REGION Network 79: Coordination Out - Decoilers Horizontal Rotation
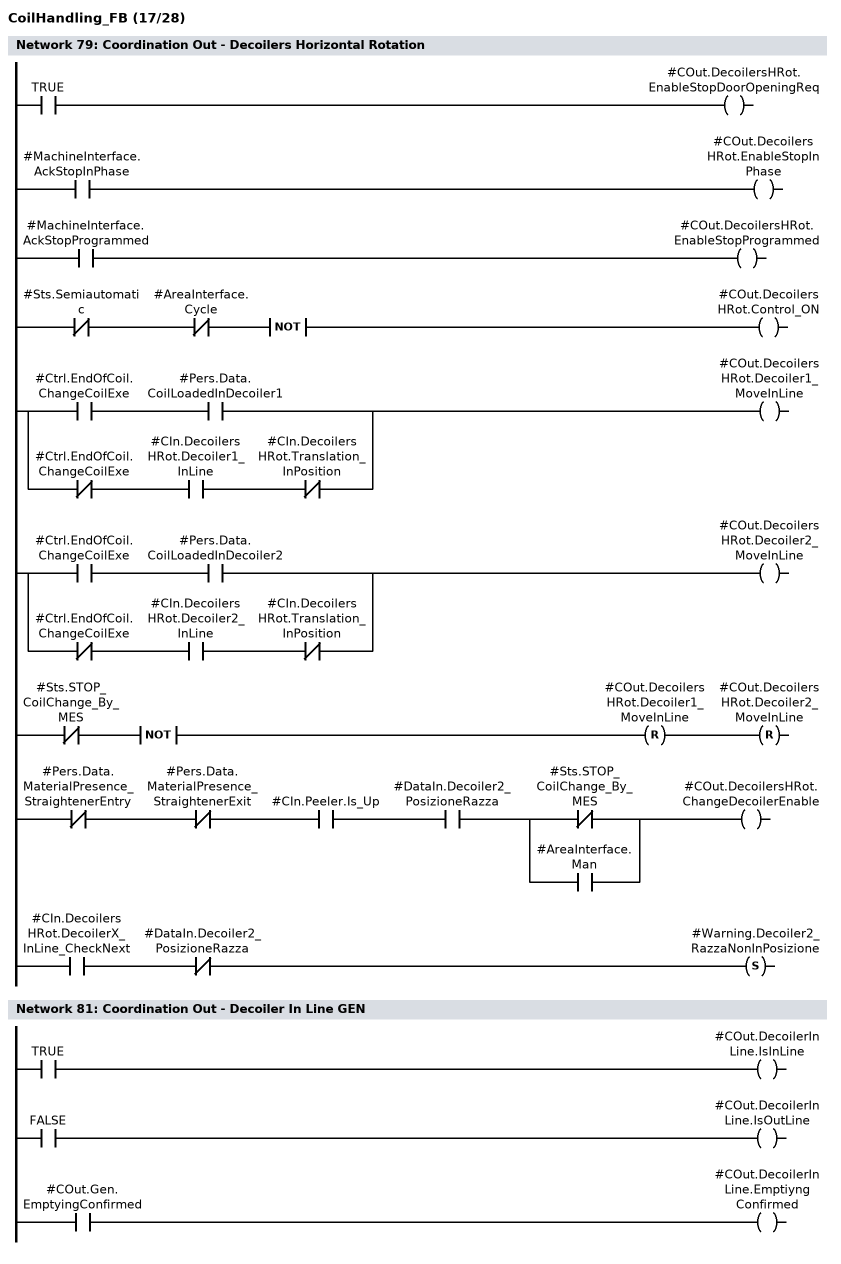
   RUNG wire#powerrail
      Contact( TRUE )
      Coil( #COut.DecoilersHRot.EnableStopDoorOpeningReq )
   END_RUNG
   RUNG wire#powerrail
      Contact( #MachineInterface.AckStopInPhase )
      Coil( #COut.DecoilersHRot.EnableStopInPhase )
   END_RUNG
   RUNG wire#powerrail
      Contact( #MachineInterface.AckStopProgrammed )
      Coil( #COut.DecoilersHRot.EnableStopProgrammed )
   END_RUNG
   RUNG wire#powerrail
      I_Contact( #Sts.Semiautomatic )
      I_Contact( #AreaInterface.Cycle )
      Not()
      Coil( #COut.DecoilersHRot.Control_ON )
   END_RUNG
   RUNG wire#powerrail
      Contact( #Ctrl.EndOfCoil.ChangeCoilExe )
      Contact( #Pers.Data.CoilLoadedInDecoiler1 )
      wire#w1
      Coil( #COut.DecoilersHRot.Decoiler1_MoveInLine )
   END_RUNG
   RUNG wire#powerrail
      I_Contact( #Ctrl.EndOfCoil.ChangeCoilExe )
      Contact( #CIn.DecoilersHRot.Decoiler1_InLine )
      I_Contact( #CIn.DecoilersHRot.Translation_InPosition )
   END_RUNG wire#w1
   RUNG wire#powerrail
      Contact( #Ctrl.EndOfCoil.ChangeCoilExe )
      Contact( #Pers.Data.CoilLoadedInDecoiler2 )
      wire#w2
      Coil( #COut.DecoilersHRot.Decoiler2_MoveInLine )
   END_RUNG
   RUNG wire#powerrail
      I_Contact( #Ctrl.EndOfCoil.ChangeCoilExe )
      Contact( #CIn.DecoilersHRot.Decoiler2_InLine )
      I_Contact( #CIn.DecoilersHRot.Translation_InPosition )
   END_RUNG wire#w2
   RUNG wire#powerrail
      I_Contact( #Sts.STOP_CoilChange_By_MES )
      Not()
      R_Coil( #COut.DecoilersHRot.Decoiler1_MoveInLine )
      R_Coil( #COut.DecoilersHRot.Decoiler2_MoveInLine )
   END_RUNG
   RUNG wire#powerrail
      I_Contact( #Pers.Data.MaterialPresence_StraightenerEntry )
      I_Contact( #Pers.Data.MaterialPresence_StraightenerExit )
      Contact( #CIn.Peeler.Is_Up )
      Contact( #DataIn.Decoiler2_PosizioneRazza )
      wire#w3
      I_Contact( #Sts.STOP_CoilChange_By_MES )
      wire#w4
      Coil( #COut.DecoilersHRot.ChangeDecoilerEnable )
   END_RUNG
   RUNG wire#w3
      Contact( #AreaInterface.Man )
   END_RUNG wire#w4
   RUNG wire#powerrail
      Contact( #CIn.DecoilersHRot.DecoilerX_InLine_CheckNext )
      I_Contact( #DataIn.Decoiler2_PosizioneRazza )
      S_Coil( #Warning.Decoiler2_RazzaNonInPosizione )
   END_RUNG
   // the same network as SCL:
   #COut.DecoilersHRot.EnableStopDoorOpeningReq := TRUE;
   #COut.DecoilersHRot.EnableStopInPhase := #MachineInterface.AckStopInPhase;
   #COut.DecoilersHRot.EnableStopProgrammed := #MachineInterface.AckStopProgrammed;
   #COut.DecoilersHRot.Control_ON := NOT (NOT #Sts.Semiautomatic AND NOT #AreaInterface.Cycle);
   #COut.DecoilersHRot.Decoiler1_MoveInLine := (#Ctrl.EndOfCoil.ChangeCoilExe AND #Pers.Data.CoilLoadedInDecoiler1) OR (NOT #Ctrl.EndOfCoil.ChangeCoilExe AND #CIn.DecoilersHRot.Decoiler1_InLine AND NOT #CIn.DecoilersHRot.Translation_InPosition);
   #COut.DecoilersHRot.Decoiler2_MoveInLine := (#Ctrl.EndOfCoil.ChangeCoilExe AND #Pers.Data.CoilLoadedInDecoiler2) OR (NOT #Ctrl.EndOfCoil.ChangeCoilExe AND #CIn.DecoilersHRot.Decoiler2_InLine AND NOT #CIn.DecoilersHRot.Translation_InPosition);
   IF NOT (NOT #Sts.STOP_CoilChange_By_MES) THEN
       #COut.DecoilersHRot.Decoiler1_MoveInLine := FALSE;
       #COut.DecoilersHRot.Decoiler2_MoveInLine := FALSE;
   END_IF;
   #COut.DecoilersHRot.ChangeDecoilerEnable := NOT #Pers.Data.MaterialPresence_StraightenerEntry AND NOT #Pers.Data.MaterialPresence_StraightenerExit AND #CIn.Peeler.Is_Up AND #DataIn.Decoiler2_PosizioneRazza AND (NOT #Sts.STOP_CoilChange_By_MES OR #AreaInterface.Man);
   IF #CIn.DecoilersHRot.DecoilerX_InLine_CheckNext AND NOT #DataIn.Decoiler2_PosizioneRazza THEN
       #Warning.Decoiler2_RazzaNonInPosizione := TRUE;
   END_IF;
END_REGION

REGION Network 80: <+>
END_REGION

REGION Network 81: Coordination Out - Decoiler In Line GEN
   RUNG wire#powerrail
      Contact( TRUE )
      Coil( #COut.DecoilerInLine.IsInLine )
   END_RUNG
   RUNG wire#powerrail
      Contact( FALSE )
      Coil( #COut.DecoilerInLine.IsOutLine )
   END_RUNG
   RUNG wire#powerrail
      Contact( #COut.Gen.EmptyingConfirmed )
      Coil( #COut.DecoilerInLine.EmptiyngConfirmed )
   END_RUNG
   // the same network as SCL:
   #COut.DecoilerInLine.IsInLine := TRUE;
   #COut.DecoilerInLine.IsOutLine := FALSE;
   #COut.DecoilerInLine.EmptiyngConfirmed := #COut.Gen.EmptyingConfirmed;
END_REGION

REGION Network 82: Coordination Out - Decoiler in Line BRAKE
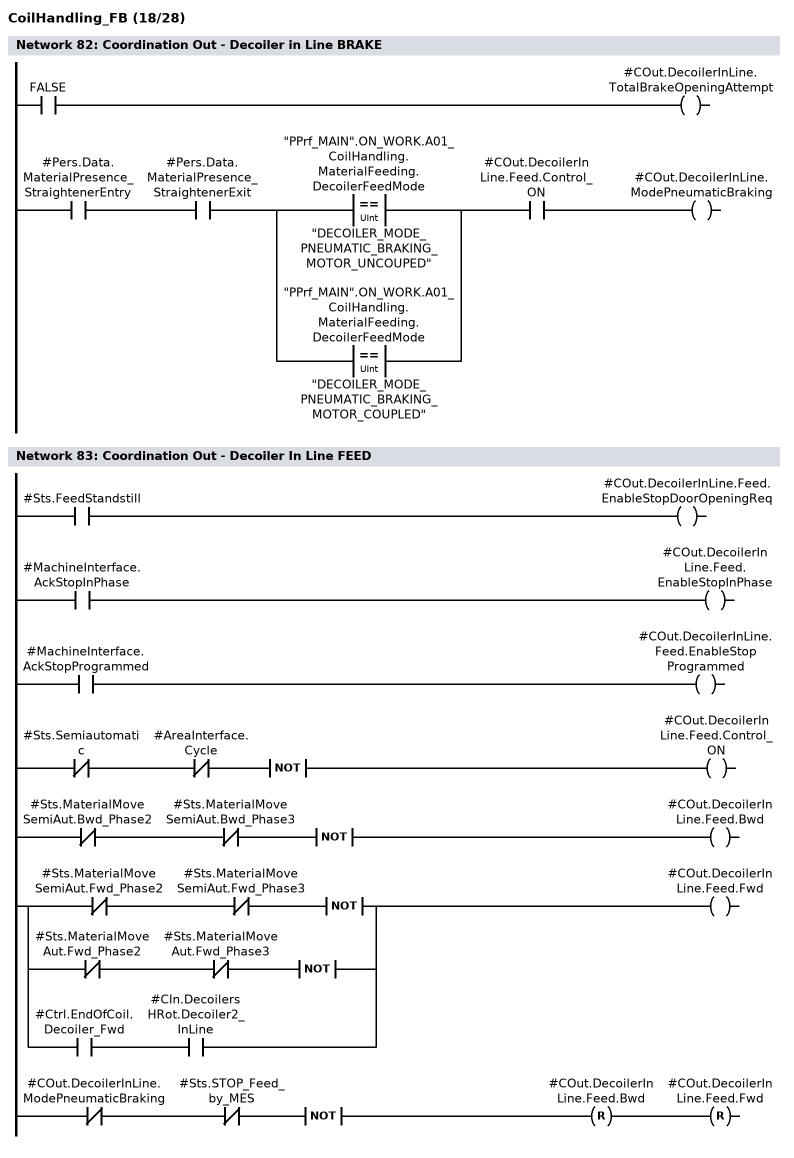
   RUNG wire#powerrail
      Contact( FALSE )
      Coil( #COut.DecoilerInLine.TotalBrakeOpeningAttempt )
   END_RUNG
   RUNG wire#powerrail
      Contact( #Pers.Data.MaterialPresence_StraightenerEntry )
      Contact( #Pers.Data.MaterialPresence_StraightenerExit )
      wire#w1
      { S7_Templates := "SrcType := UInt" } EQ_Contact(in1 := "PPrf_MAIN".ON_WORK.A01_CoilHandling.MaterialFeeding.DecoilerFeedMode, in2 := "DECOILER_MODE_PNEUMATIC_BRAKING_MOTOR_UNCOUPED")
      wire#w2
      Contact( #COut.DecoilerInLine.Feed.Control_ON )
      Coil( #COut.DecoilerInLine.ModePneumaticBraking )
   END_RUNG
   RUNG wire#w1
      { S7_Templates := "SrcType := UInt" } EQ_Contact(in1 := "PPrf_MAIN".ON_WORK.A01_CoilHandling.MaterialFeeding.DecoilerFeedMode, in2 := "DECOILER_MODE_PNEUMATIC_BRAKING_MOTOR_COUPLED")
   END_RUNG wire#w2
   // the same network as SCL:
   #COut.DecoilerInLine.TotalBrakeOpeningAttempt := FALSE;
   #COut.DecoilerInLine.ModePneumaticBraking := #Pers.Data.MaterialPresence_StraightenerEntry AND #Pers.Data.MaterialPresence_StraightenerExit AND (("PPrf_MAIN".ON_WORK.A01_CoilHandling.MaterialFeeding.DecoilerFeedMode = "DECOILER_MODE_PNEUMATIC_BRAKING_MOTOR_UNCOUPED") OR ("PPrf_MAIN".ON_WORK.A01_CoilHandling.MaterialFeeding.DecoilerFeedMode = "DECOILER_MODE_PNEUMATIC_BRAKING_MOTOR_COUPLED")) AND #COut.DecoilerInLine.Feed.Control_ON;
END_REGION

REGION Network 83: Coordination Out - Decoiler In Line FEED
   RUNG wire#powerrail
      Contact( #Sts.FeedStandstill )
      Coil( #COut.DecoilerInLine.Feed.EnableStopDoorOpeningReq )
   END_RUNG
   RUNG wire#powerrail
      Contact( #MachineInterface.AckStopInPhase )
      Coil( #COut.DecoilerInLine.Feed.EnableStopInPhase )
   END_RUNG
   RUNG wire#powerrail
      Contact( #MachineInterface.AckStopProgrammed )
      Coil( #COut.DecoilerInLine.Feed.EnableStopProgrammed )
   END_RUNG
   RUNG wire#powerrail
      I_Contact( #Sts.Semiautomatic )
      I_Contact( #AreaInterface.Cycle )
      Not()
      Coil( #COut.DecoilerInLine.Feed.Control_ON )
   END_RUNG
   RUNG wire#powerrail
      I_Contact( #Sts.MaterialMoveSemiAut.Bwd_Phase2 )
      I_Contact( #Sts.MaterialMoveSemiAut.Bwd_Phase3 )
      Not()
      Coil( #COut.DecoilerInLine.Feed.Bwd )
   END_RUNG
   RUNG wire#powerrail
      I_Contact( #Sts.MaterialMoveSemiAut.Fwd_Phase2 )
      I_Contact( #Sts.MaterialMoveSemiAut.Fwd_Phase3 )
      Not()
      wire#w1
      Coil( #COut.DecoilerInLine.Feed.Fwd )
   END_RUNG
   RUNG wire#powerrail
      I_Contact( #Sts.MaterialMoveAut.Fwd_Phase2 )
      I_Contact( #Sts.MaterialMoveAut.Fwd_Phase3 )
      Not()
   END_RUNG wire#w1
   RUNG wire#powerrail
      Contact( #Ctrl.EndOfCoil.Decoiler_Fwd )
      Contact( #CIn.DecoilersHRot.Decoiler2_InLine )
   END_RUNG wire#w1
   RUNG wire#powerrail
      I_Contact( #COut.DecoilerInLine.ModePneumaticBraking )
      I_Contact( #Sts.STOP_Feed_by_MES )
      Not()
      R_Coil( #COut.DecoilerInLine.Feed.Bwd )
      R_Coil( #COut.DecoilerInLine.Feed.Fwd )
   END_RUNG
   // the same network as SCL:
   #COut.DecoilerInLine.Feed.EnableStopDoorOpeningReq := #Sts.FeedStandstill;
   #COut.DecoilerInLine.Feed.EnableStopInPhase := #MachineInterface.AckStopInPhase;
   #COut.DecoilerInLine.Feed.EnableStopProgrammed := #MachineInterface.AckStopProgrammed;
   #COut.DecoilerInLine.Feed.Control_ON := NOT (NOT #Sts.Semiautomatic AND NOT #AreaInterface.Cycle);
   #COut.DecoilerInLine.Feed.Bwd := NOT (NOT #Sts.MaterialMoveSemiAut.Bwd_Phase2 AND NOT #Sts.MaterialMoveSemiAut.Bwd_Phase3);
   #COut.DecoilerInLine.Feed.Fwd := NOT (NOT #Sts.MaterialMoveSemiAut.Fwd_Phase2 AND NOT #Sts.MaterialMoveSemiAut.Fwd_Phase3) OR NOT (NOT #Sts.MaterialMoveAut.Fwd_Phase2 AND NOT #Sts.MaterialMoveAut.Fwd_Phase3) OR (#Ctrl.EndOfCoil.Decoiler_Fwd AND #CIn.DecoilersHRot.Decoiler2_InLine);
   IF NOT (NOT #COut.DecoilerInLine.ModePneumaticBraking AND NOT #Sts.STOP_Feed_by_MES) THEN
       #COut.DecoilerInLine.Feed.Bwd := FALSE;
       #COut.DecoilerInLine.Feed.Fwd := FALSE;
   END_IF;
END_REGION

REGION Network 84: Coordination Out - Decoiler in Line COUPLING
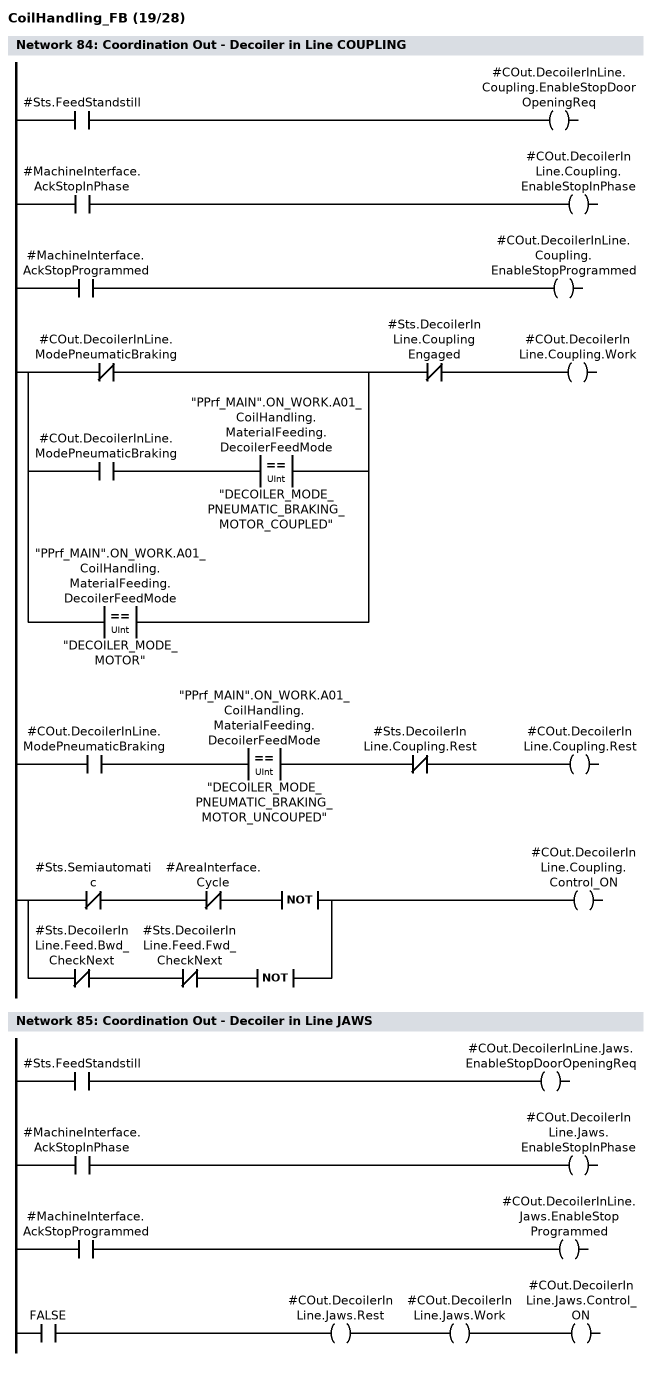
   RUNG wire#powerrail
      Contact( #Sts.FeedStandstill )
      Coil( #COut.DecoilerInLine.Coupling.EnableStopDoorOpeningReq )
   END_RUNG
   RUNG wire#powerrail
      Contact( #MachineInterface.AckStopInPhase )
      Coil( #COut.DecoilerInLine.Coupling.EnableStopInPhase )
   END_RUNG
   RUNG wire#powerrail
      Contact( #MachineInterface.AckStopProgrammed )
      Coil( #COut.DecoilerInLine.Coupling.EnableStopProgrammed )
   END_RUNG
   RUNG wire#powerrail
      I_Contact( #COut.DecoilerInLine.ModePneumaticBraking )
      wire#w1
      I_Contact( #Sts.DecoilerInLine.CouplingEngaged )
      Coil( #COut.DecoilerInLine.Coupling.Work )
   END_RUNG
   RUNG wire#powerrail
      Contact( #COut.DecoilerInLine.ModePneumaticBraking )
      { S7_Templates := "SrcType := UInt" } EQ_Contact(in1 := "PPrf_MAIN".ON_WORK.A01_CoilHandling.MaterialFeeding.DecoilerFeedMode, in2 := "DECOILER_MODE_PNEUMATIC_BRAKING_MOTOR_COUPLED")
   END_RUNG wire#w1
   RUNG wire#powerrail
      { S7_Templates := "SrcType := UInt" } EQ_Contact(in1 := "PPrf_MAIN".ON_WORK.A01_CoilHandling.MaterialFeeding.DecoilerFeedMode, in2 := "DECOILER_MODE_MOTOR")
   END_RUNG wire#w1
   RUNG wire#powerrail
      Contact( #COut.DecoilerInLine.ModePneumaticBraking )
      { S7_Templates := "SrcType := UInt" } EQ_Contact(in1 := "PPrf_MAIN".ON_WORK.A01_CoilHandling.MaterialFeeding.DecoilerFeedMode, in2 := "DECOILER_MODE_PNEUMATIC_BRAKING_MOTOR_UNCOUPED")
      I_Contact( #Sts.DecoilerInLine.Coupling.Rest )
      Coil( #COut.DecoilerInLine.Coupling.Rest )
   END_RUNG
   RUNG wire#powerrail
      I_Contact( #Sts.Semiautomatic )
      I_Contact( #AreaInterface.Cycle )
      Not()
      wire#w2
      Coil( #COut.DecoilerInLine.Coupling.Control_ON )
   END_RUNG
   RUNG wire#powerrail
      I_Contact( #Sts.DecoilerInLine.Feed.Bwd_CheckNext )
      I_Contact( #Sts.DecoilerInLine.Feed.Fwd_CheckNext )
      Not()
   END_RUNG wire#w2
   // the same network as SCL:
   #COut.DecoilerInLine.Coupling.EnableStopDoorOpeningReq := #Sts.FeedStandstill;
   #COut.DecoilerInLine.Coupling.EnableStopInPhase := #MachineInterface.AckStopInPhase;
   #COut.DecoilerInLine.Coupling.EnableStopProgrammed := #MachineInterface.AckStopProgrammed;
   #COut.DecoilerInLine.Coupling.Work := (NOT #COut.DecoilerInLine.ModePneumaticBraking OR (#COut.DecoilerInLine.ModePneumaticBraking AND ("PPrf_MAIN".ON_WORK.A01_CoilHandling.MaterialFeeding.DecoilerFeedMode = "DECOILER_MODE_PNEUMATIC_BRAKING_MOTOR_COUPLED")) OR ("PPrf_MAIN".ON_WORK.A01_CoilHandling.MaterialFeeding.DecoilerFeedMode = "DECOILER_MODE_MOTOR")) AND NOT #Sts.DecoilerInLine.CouplingEngaged;
   #COut.DecoilerInLine.Coupling.Rest := #COut.DecoilerInLine.ModePneumaticBraking AND ("PPrf_MAIN".ON_WORK.A01_CoilHandling.MaterialFeeding.DecoilerFeedMode = "DECOILER_MODE_PNEUMATIC_BRAKING_MOTOR_UNCOUPED") AND NOT #Sts.DecoilerInLine.Coupling.Rest;
   #COut.DecoilerInLine.Coupling.Control_ON := NOT (NOT #Sts.Semiautomatic AND NOT #AreaInterface.Cycle) OR NOT (NOT #Sts.DecoilerInLine.Feed.Bwd_CheckNext AND NOT #Sts.DecoilerInLine.Feed.Fwd_CheckNext);
END_REGION

REGION Network 85: Coordination Out - Decoiler in Line JAWS
   RUNG wire#powerrail
      Contact( #Sts.FeedStandstill )
      Coil( #COut.DecoilerInLine.Jaws.EnableStopDoorOpeningReq )
   END_RUNG
   RUNG wire#powerrail
      Contact( #MachineInterface.AckStopInPhase )
      Coil( #COut.DecoilerInLine.Jaws.EnableStopInPhase )
   END_RUNG
   RUNG wire#powerrail
      Contact( #MachineInterface.AckStopProgrammed )
      Coil( #COut.DecoilerInLine.Jaws.EnableStopProgrammed )
   END_RUNG
   RUNG wire#powerrail
      Contact( FALSE )
      Coil( #COut.DecoilerInLine.Jaws.Rest )
      Coil( #COut.DecoilerInLine.Jaws.Work )
      Coil( #COut.DecoilerInLine.Jaws.Control_ON )
   END_RUNG
   // the same network as SCL:
   #COut.DecoilerInLine.Jaws.EnableStopDoorOpeningReq := #Sts.FeedStandstill;
   #COut.DecoilerInLine.Jaws.EnableStopInPhase := #MachineInterface.AckStopInPhase;
   #COut.DecoilerInLine.Jaws.EnableStopProgrammed := #MachineInterface.AckStopProgrammed;
   #COut.DecoilerInLine.Jaws.Rest := FALSE;
   #COut.DecoilerInLine.Jaws.Work := FALSE;
   #COut.DecoilerInLine.Jaws.Control_ON := FALSE;
END_REGION

REGION Network 86: Coordination Out - Decoiler in Line SNUBBER
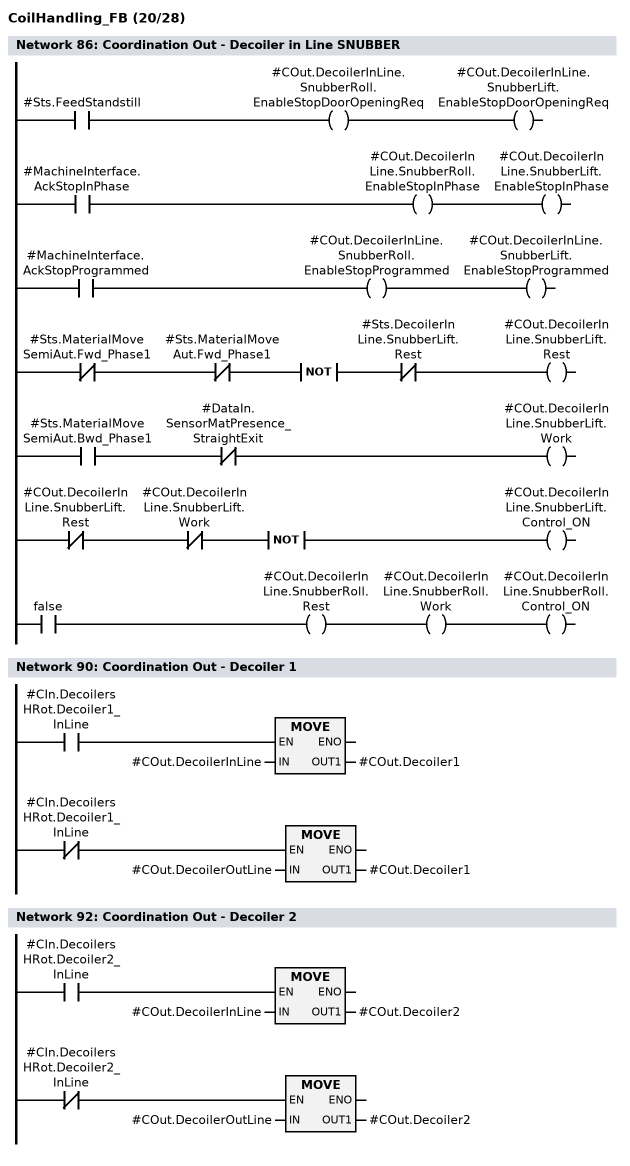
   RUNG wire#powerrail
      Contact( #Sts.FeedStandstill )
      Coil( #COut.DecoilerInLine.SnubberRoll.EnableStopDoorOpeningReq )
      Coil( #COut.DecoilerInLine.SnubberLift.EnableStopDoorOpeningReq )
   END_RUNG
   RUNG wire#powerrail
      Contact( #MachineInterface.AckStopInPhase )
      Coil( #COut.DecoilerInLine.SnubberRoll.EnableStopInPhase )
      Coil( #COut.DecoilerInLine.SnubberLift.EnableStopInPhase )
   END_RUNG
   RUNG wire#powerrail
      Contact( #MachineInterface.AckStopProgrammed )
      Coil( #COut.DecoilerInLine.SnubberRoll.EnableStopProgrammed )
      Coil( #COut.DecoilerInLine.SnubberLift.EnableStopProgrammed )
   END_RUNG
   RUNG wire#powerrail
      I_Contact( #Sts.MaterialMoveSemiAut.Fwd_Phase1 )
      I_Contact( #Sts.MaterialMoveAut.Fwd_Phase1 )
      Not()
      I_Contact( #Sts.DecoilerInLine.SnubberLift.Rest )
      Coil( #COut.DecoilerInLine.SnubberLift.Rest )
   END_RUNG
   RUNG wire#powerrail
      Contact( #Sts.MaterialMoveSemiAut.Bwd_Phase1 )
      I_Contact( #DataIn.SensorMatPresence_StraightExit )
      Coil( #COut.DecoilerInLine.SnubberLift.Work )
   END_RUNG
   RUNG wire#powerrail
      I_Contact( #COut.DecoilerInLine.SnubberLift.Rest )
      I_Contact( #COut.DecoilerInLine.SnubberLift.Work )
      Not()
      Coil( #COut.DecoilerInLine.SnubberLift.Control_ON )
   END_RUNG
   RUNG wire#powerrail
      Contact( false )
      Coil( #COut.DecoilerInLine.SnubberRoll.Rest )
      Coil( #COut.DecoilerInLine.SnubberRoll.Work )
      Coil( #COut.DecoilerInLine.SnubberRoll.Control_ON )
   END_RUNG
   // the same network as SCL:
   #COut.DecoilerInLine.SnubberRoll.EnableStopDoorOpeningReq := #Sts.FeedStandstill;
   #COut.DecoilerInLine.SnubberLift.EnableStopDoorOpeningReq := #Sts.FeedStandstill;
   #COut.DecoilerInLine.SnubberRoll.EnableStopInPhase := #MachineInterface.AckStopInPhase;
   #COut.DecoilerInLine.SnubberLift.EnableStopInPhase := #MachineInterface.AckStopInPhase;
   #COut.DecoilerInLine.SnubberRoll.EnableStopProgrammed := #MachineInterface.AckStopProgrammed;
   #COut.DecoilerInLine.SnubberLift.EnableStopProgrammed := #MachineInterface.AckStopProgrammed;
   #COut.DecoilerInLine.SnubberLift.Rest := NOT (NOT #Sts.MaterialMoveSemiAut.Fwd_Phase1 AND NOT #Sts.MaterialMoveAut.Fwd_Phase1) AND NOT #Sts.DecoilerInLine.SnubberLift.Rest;
   #COut.DecoilerInLine.SnubberLift.Work := #Sts.MaterialMoveSemiAut.Bwd_Phase1 AND NOT #DataIn.SensorMatPresence_StraightExit;
   #COut.DecoilerInLine.SnubberLift.Control_ON := NOT (NOT #COut.DecoilerInLine.SnubberLift.Rest AND NOT #COut.DecoilerInLine.SnubberLift.Work);
   #COut.DecoilerInLine.SnubberRoll.Rest := false;
   #COut.DecoilerInLine.SnubberRoll.Work := false;
   #COut.DecoilerInLine.SnubberRoll.Control_ON := false;
END_REGION

REGION Network 87: <+>
END_REGION

REGION Network 88 (SCL): Coordination Out - Decoiler Out ofLine
   #COut.DecoilerOutLine.IsOutLine := TRUE;
   #COut.DecoilerOutLine.IsInLine := FALSE;

   #COut.DecoilerOutLine.ModePneumaticBraking := FALSE;
   #COut.DecoilerOutLine.TotalBrakeOpeningAttempt := FALSE;
   #COut.DecoilerOutLine.EmptiyngConfirmed := FALSE;

   #COut.DecoilerOutLine.Feed.Control_ON := FALSE;
   #COut.DecoilerOutLine.Feed.Bwd := FALSE;
   #COut.DecoilerOutLine.Feed.Fwd := FALSE;

   #COut.DecoilerOutLine.Jaws.Control_ON := FALSE;
   #COut.DecoilerOutLine.Jaws.Rest := FALSE;
   #COut.DecoilerOutLine.Jaws.Work := FALSE;

   #COut.DecoilerOutLine.Coupling.Control_ON := FALSE;
   #COut.DecoilerOutLine.Coupling.Rest := FALSE;
   #COut.DecoilerOutLine.Coupling.Work := FALSE;

   #COut.DecoilerOutLine.SnubberLift.Control_ON := FALSE;
   #COut.DecoilerOutLine.SnubberLift.Rest := FALSE;
   #COut.DecoilerOutLine.SnubberLift.Work := FALSE;

   #COut.DecoilerOutLine.SnubberRoll.Control_ON := FALSE;
   #COut.DecoilerOutLine.SnubberRoll.Rest := FALSE;
   #COut.DecoilerOutLine.SnubberRoll.Work := FALSE;
END_REGION

REGION Network 89: <+>
END_REGION

REGION Network 90: Coordination Out - Decoiler 1
   RUNG wire#powerrail
      Contact( #CIn.DecoilersHRot.Decoiler1_InLine )
      Move(in := #COut.DecoilerInLine, out1 => #COut.Decoiler1)
   END_RUNG
   RUNG wire#powerrail
      I_Contact( #CIn.DecoilersHRot.Decoiler1_InLine )
      Move(in := #COut.DecoilerOutLine, out1 => #COut.Decoiler1)
   END_RUNG
   // the same network as SCL:
   IF #CIn.DecoilersHRot.Decoiler1_InLine THEN #COut.Decoiler1 := #COut.DecoilerInLine; END_IF;
   IF NOT #CIn.DecoilersHRot.Decoiler1_InLine THEN #COut.Decoiler1 := #COut.DecoilerOutLine; END_IF;
END_REGION

REGION Network 91: <+>
END_REGION

REGION Network 92: Coordination Out - Decoiler 2
   RUNG wire#powerrail
      Contact( #CIn.DecoilersHRot.Decoiler2_InLine )
      Move(in := #COut.DecoilerInLine, out1 => #COut.Decoiler2)
   END_RUNG
   RUNG wire#powerrail
      I_Contact( #CIn.DecoilersHRot.Decoiler2_InLine )
      Move(in := #COut.DecoilerOutLine, out1 => #COut.Decoiler2)
   END_RUNG
   // the same network as SCL:
   IF #CIn.DecoilersHRot.Decoiler2_InLine THEN #COut.Decoiler2 := #COut.DecoilerInLine; END_IF;
   IF NOT #CIn.DecoilersHRot.Decoiler2_InLine THEN #COut.Decoiler2 := #COut.DecoilerOutLine; END_IF;
END_REGION

REGION Network 93: <+>
END_REGION

REGION Network 94: Coordination Out - Peelers
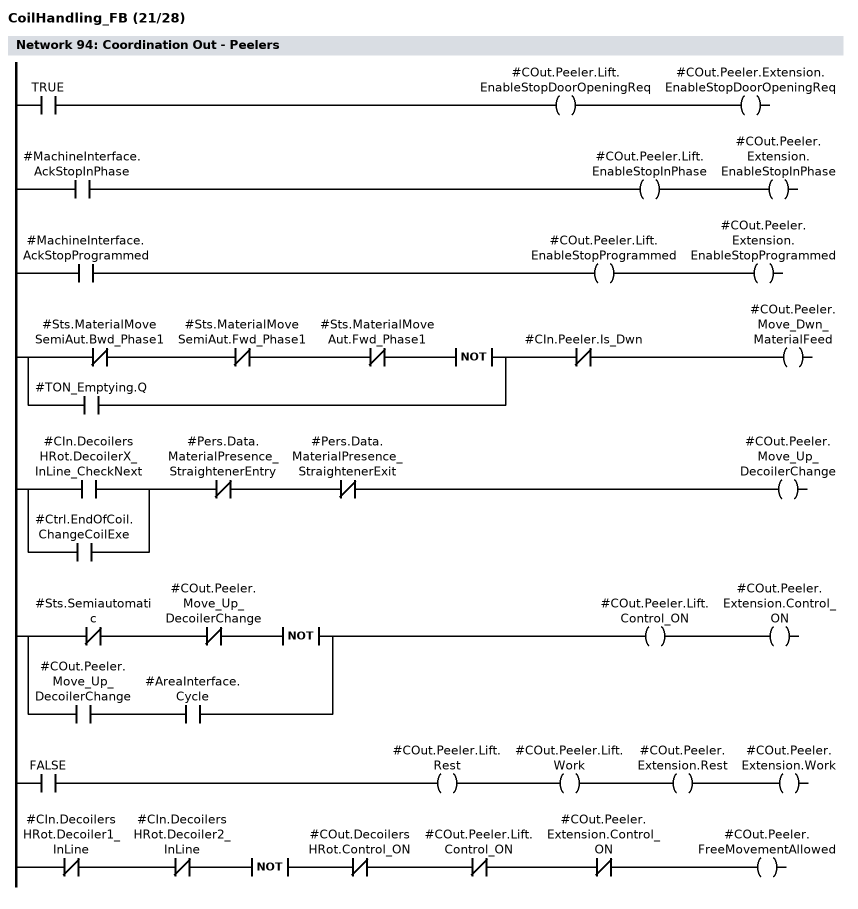
   RUNG wire#powerrail
      Contact( TRUE )
      Coil( #COut.Peeler.Lift.EnableStopDoorOpeningReq )
      Coil( #COut.Peeler.Extension.EnableStopDoorOpeningReq )
   END_RUNG
   RUNG wire#powerrail
      Contact( #MachineInterface.AckStopInPhase )
      Coil( #COut.Peeler.Lift.EnableStopInPhase )
      Coil( #COut.Peeler.Extension.EnableStopInPhase )
   END_RUNG
   RUNG wire#powerrail
      Contact( #MachineInterface.AckStopProgrammed )
      Coil( #COut.Peeler.Lift.EnableStopProgrammed )
      Coil( #COut.Peeler.Extension.EnableStopProgrammed )
   END_RUNG
   RUNG wire#powerrail
      I_Contact( #Sts.MaterialMoveSemiAut.Bwd_Phase1 )
      I_Contact( #Sts.MaterialMoveSemiAut.Fwd_Phase1 )
      I_Contact( #Sts.MaterialMoveAut.Fwd_Phase1 )
      Not()
      wire#w1
      I_Contact( #CIn.Peeler.Is_Dwn )
      Coil( #COut.Peeler.Move_Dwn_MaterialFeed )
   END_RUNG
   RUNG wire#powerrail
      Contact( #TON_Emptying.Q )
   END_RUNG wire#w1
   RUNG wire#powerrail
      Contact( #CIn.DecoilersHRot.DecoilerX_InLine_CheckNext )
      wire#w2
      I_Contact( #Pers.Data.MaterialPresence_StraightenerEntry )
      I_Contact( #Pers.Data.MaterialPresence_StraightenerExit )
      Coil( #COut.Peeler.Move_Up_DecoilerChange )
   END_RUNG
   RUNG wire#powerrail
      Contact( #Ctrl.EndOfCoil.ChangeCoilExe )
   END_RUNG wire#w2
   RUNG wire#powerrail
      I_Contact( #Sts.Semiautomatic )
      I_Contact( #COut.Peeler.Move_Up_DecoilerChange )
      Not()
      wire#w3
      Coil( #COut.Peeler.Lift.Control_ON )
      Coil( #COut.Peeler.Extension.Control_ON )
   END_RUNG
   RUNG wire#powerrail
      Contact( #COut.Peeler.Move_Up_DecoilerChange )
      Contact( #AreaInterface.Cycle )
   END_RUNG wire#w3
   RUNG wire#powerrail
      Contact( FALSE )
      Coil( #COut.Peeler.Lift.Rest )
      Coil( #COut.Peeler.Lift.Work )
      Coil( #COut.Peeler.Extension.Rest )
      Coil( #COut.Peeler.Extension.Work )
   END_RUNG
   RUNG wire#powerrail
      I_Contact( #CIn.DecoilersHRot.Decoiler1_InLine )
      I_Contact( #CIn.DecoilersHRot.Decoiler2_InLine )
      Not()
      I_Contact( #COut.DecoilersHRot.Control_ON )
      I_Contact( #COut.Peeler.Lift.Control_ON )
      I_Contact( #COut.Peeler.Extension.Control_ON )
      Coil( #COut.Peeler.FreeMovementAllowed )
   END_RUNG
   // the same network as SCL:
   #COut.Peeler.Lift.EnableStopDoorOpeningReq := TRUE;
   #COut.Peeler.Extension.EnableStopDoorOpeningReq := TRUE;
   #COut.Peeler.Lift.EnableStopInPhase := #MachineInterface.AckStopInPhase;
   #COut.Peeler.Extension.EnableStopInPhase := #MachineInterface.AckStopInPhase;
   #COut.Peeler.Lift.EnableStopProgrammed := #MachineInterface.AckStopProgrammed;
   #COut.Peeler.Extension.EnableStopProgrammed := #MachineInterface.AckStopProgrammed;
   #COut.Peeler.Move_Dwn_MaterialFeed := (NOT (NOT #Sts.MaterialMoveSemiAut.Bwd_Phase1 AND NOT #Sts.MaterialMoveSemiAut.Fwd_Phase1 AND NOT #Sts.MaterialMoveAut.Fwd_Phase1) OR #TON_Emptying.Q) AND NOT #CIn.Peeler.Is_Dwn;
   #COut.Peeler.Move_Up_DecoilerChange := (#CIn.DecoilersHRot.DecoilerX_InLine_CheckNext OR #Ctrl.EndOfCoil.ChangeCoilExe) AND NOT #Pers.Data.MaterialPresence_StraightenerEntry AND NOT #Pers.Data.MaterialPresence_StraightenerExit;
   #COut.Peeler.Lift.Control_ON := NOT (NOT #Sts.Semiautomatic AND NOT #COut.Peeler.Move_Up_DecoilerChange) OR (#COut.Peeler.Move_Up_DecoilerChange AND #AreaInterface.Cycle);
   #COut.Peeler.Extension.Control_ON := #COut.Peeler.Lift.Control_ON;
   #COut.Peeler.Lift.Rest := FALSE;
   #COut.Peeler.Lift.Work := FALSE;
   #COut.Peeler.Extension.Rest := FALSE;
   #COut.Peeler.Extension.Work := FALSE;
   #COut.Peeler.FreeMovementAllowed := NOT (NOT #CIn.DecoilersHRot.Decoiler1_InLine AND NOT #CIn.DecoilersHRot.Decoiler2_InLine) AND NOT #COut.DecoilersHRot.Control_ON AND NOT #COut.Peeler.Lift.Control_ON AND NOT #COut.Peeler.Extension.Control_ON;
END_REGION

REGION Network 95: <+>
END_REGION

REGION Network 96: Coordination Out - Straightener FEED
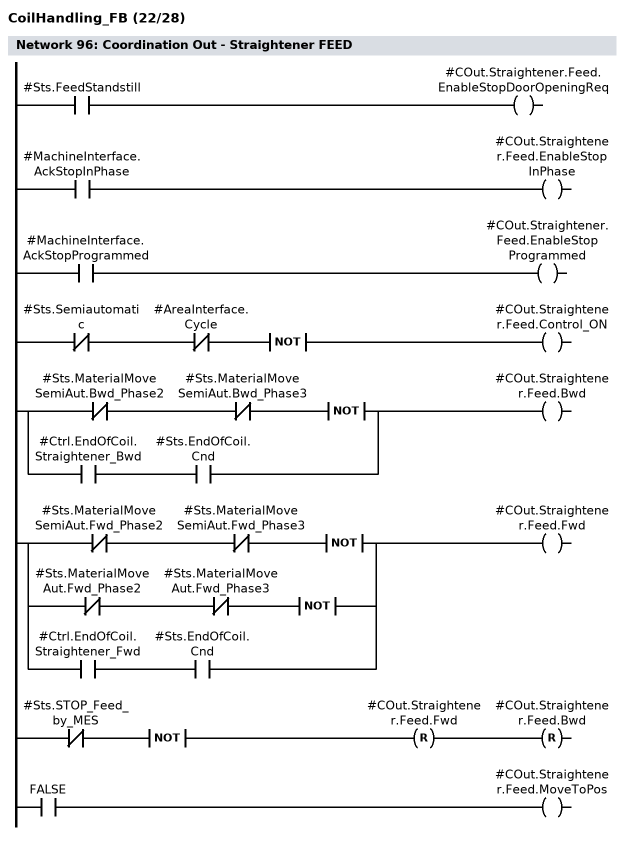
   RUNG wire#powerrail
      Contact( #Sts.FeedStandstill )
      Coil( #COut.Straightener.Feed.EnableStopDoorOpeningReq )
   END_RUNG
   RUNG wire#powerrail
      Contact( #MachineInterface.AckStopInPhase )
      Coil( #COut.Straightener.Feed.EnableStopInPhase )
   END_RUNG
   RUNG wire#powerrail
      Contact( #MachineInterface.AckStopProgrammed )
      Coil( #COut.Straightener.Feed.EnableStopProgrammed )
   END_RUNG
   RUNG wire#powerrail
      I_Contact( #Sts.Semiautomatic )
      I_Contact( #AreaInterface.Cycle )
      Not()
      Coil( #COut.Straightener.Feed.Control_ON )
   END_RUNG
   RUNG wire#powerrail
      I_Contact( #Sts.MaterialMoveSemiAut.Bwd_Phase2 )
      I_Contact( #Sts.MaterialMoveSemiAut.Bwd_Phase3 )
      Not()
      wire#w1
      Coil( #COut.Straightener.Feed.Bwd )
   END_RUNG
   RUNG wire#powerrail
      Contact( #Ctrl.EndOfCoil.Straightener_Bwd )
      Contact( #Sts.EndOfCoil.Cnd )
   END_RUNG wire#w1
   RUNG wire#powerrail
      I_Contact( #Sts.MaterialMoveSemiAut.Fwd_Phase2 )
      I_Contact( #Sts.MaterialMoveSemiAut.Fwd_Phase3 )
      Not()
      wire#w2
      Coil( #COut.Straightener.Feed.Fwd )
   END_RUNG
   RUNG wire#powerrail
      I_Contact( #Sts.MaterialMoveAut.Fwd_Phase2 )
      I_Contact( #Sts.MaterialMoveAut.Fwd_Phase3 )
      Not()
   END_RUNG wire#w2
   RUNG wire#powerrail
      Contact( #Ctrl.EndOfCoil.Straightener_Fwd )
      Contact( #Sts.EndOfCoil.Cnd )
   END_RUNG wire#w2
   RUNG wire#powerrail
      I_Contact( #Sts.STOP_Feed_by_MES )
      Not()
      R_Coil( #COut.Straightener.Feed.Fwd )
      R_Coil( #COut.Straightener.Feed.Bwd )
   END_RUNG
   RUNG wire#powerrail
      Contact( FALSE )
      Coil( #COut.Straightener.Feed.MoveToPos )
   END_RUNG
   // the same network as SCL:
   #COut.Straightener.Feed.EnableStopDoorOpeningReq := #Sts.FeedStandstill;
   #COut.Straightener.Feed.EnableStopInPhase := #MachineInterface.AckStopInPhase;
   #COut.Straightener.Feed.EnableStopProgrammed := #MachineInterface.AckStopProgrammed;
   #COut.Straightener.Feed.Control_ON := NOT (NOT #Sts.Semiautomatic AND NOT #AreaInterface.Cycle);
   #COut.Straightener.Feed.Bwd := NOT (NOT #Sts.MaterialMoveSemiAut.Bwd_Phase2 AND NOT #Sts.MaterialMoveSemiAut.Bwd_Phase3) OR (#Ctrl.EndOfCoil.Straightener_Bwd AND #Sts.EndOfCoil.Cnd);
   #COut.Straightener.Feed.Fwd := NOT (NOT #Sts.MaterialMoveSemiAut.Fwd_Phase2 AND NOT #Sts.MaterialMoveSemiAut.Fwd_Phase3) OR NOT (NOT #Sts.MaterialMoveAut.Fwd_Phase2 AND NOT #Sts.MaterialMoveAut.Fwd_Phase3) OR (#Ctrl.EndOfCoil.Straightener_Fwd AND #Sts.EndOfCoil.Cnd);
   IF NOT (NOT #Sts.STOP_Feed_by_MES) THEN
       #COut.Straightener.Feed.Fwd := FALSE;
       #COut.Straightener.Feed.Bwd := FALSE;
   END_IF;
   #COut.Straightener.Feed.MoveToPos := FALSE;
END_REGION

REGION Network 97: Coordination Out - Straightener ENTRY ROLL
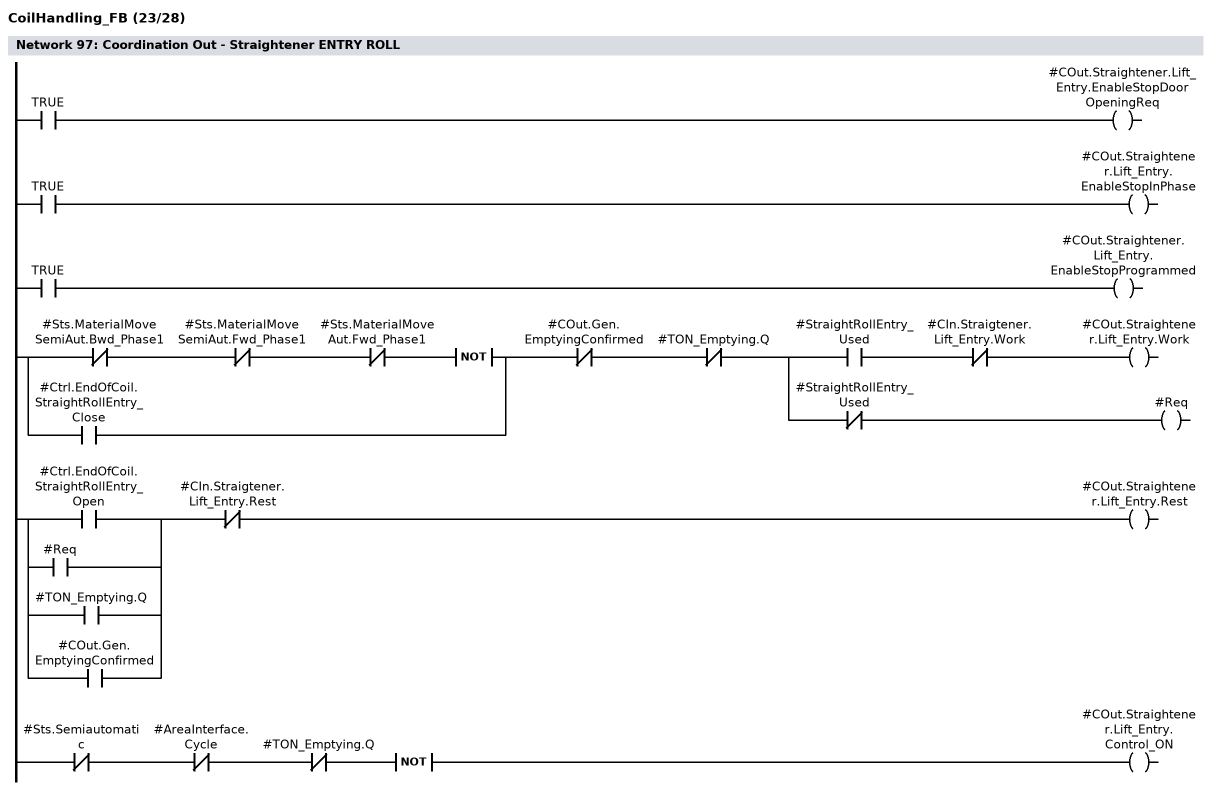
   RUNG wire#powerrail
      Contact( TRUE )
      Coil( #COut.Straightener.Lift_Entry.EnableStopDoorOpeningReq )
   END_RUNG
   RUNG wire#powerrail
      Contact( TRUE )
      Coil( #COut.Straightener.Lift_Entry.EnableStopInPhase )
   END_RUNG
   RUNG wire#powerrail
      Contact( TRUE )
      Coil( #COut.Straightener.Lift_Entry.EnableStopProgrammed )
   END_RUNG
   RUNG wire#powerrail
      I_Contact( #Sts.MaterialMoveSemiAut.Bwd_Phase1 )
      I_Contact( #Sts.MaterialMoveSemiAut.Fwd_Phase1 )
      I_Contact( #Sts.MaterialMoveAut.Fwd_Phase1 )
      Not()
      wire#w1
      I_Contact( #COut.Gen.EmptyingConfirmed )
      I_Contact( #TON_Emptying.Q )
      wire#w2
      Contact( #StraightRollEntry_Used )
      I_Contact( #CIn.Straigtener.Lift_Entry.Work )
      Coil( #COut.Straightener.Lift_Entry.Work )
   END_RUNG
   RUNG wire#powerrail
      Contact( #Ctrl.EndOfCoil.StraightRollEntry_Close )
   END_RUNG wire#w1
   RUNG wire#w2
      I_Contact( #StraightRollEntry_Used )
      Coil( #Req )
   END_RUNG
   RUNG wire#powerrail
      Contact( #Ctrl.EndOfCoil.StraightRollEntry_Open )
      wire#w3
      I_Contact( #CIn.Straigtener.Lift_Entry.Rest )
      Coil( #COut.Straightener.Lift_Entry.Rest )
   END_RUNG
   RUNG wire#powerrail
      Contact( #Req )
   END_RUNG wire#w3
   RUNG wire#powerrail
      Contact( #TON_Emptying.Q )
   END_RUNG wire#w3
   RUNG wire#powerrail
      Contact( #COut.Gen.EmptyingConfirmed )
   END_RUNG wire#w3
   RUNG wire#powerrail
      I_Contact( #Sts.Semiautomatic )
      I_Contact( #AreaInterface.Cycle )
      I_Contact( #TON_Emptying.Q )
      Not()
      Coil( #COut.Straightener.Lift_Entry.Control_ON )
   END_RUNG
   // the same network as SCL:
   #COut.Straightener.Lift_Entry.EnableStopDoorOpeningReq := TRUE;
   #COut.Straightener.Lift_Entry.EnableStopInPhase := TRUE;
   #COut.Straightener.Lift_Entry.EnableStopProgrammed := TRUE;
   #_w1 := (NOT (NOT #Sts.MaterialMoveSemiAut.Bwd_Phase1 AND NOT #Sts.MaterialMoveSemiAut.Fwd_Phase1 AND NOT #Sts.MaterialMoveAut.Fwd_Phase1) OR #Ctrl.EndOfCoil.StraightRollEntry_Close) AND NOT #COut.Gen.EmptyingConfirmed AND NOT #TON_Emptying.Q;
   #COut.Straightener.Lift_Entry.Work := #_w1 AND #StraightRollEntry_Used AND NOT #CIn.Straigtener.Lift_Entry.Work;
   #Req := #_w1 AND NOT #StraightRollEntry_Used;
   #COut.Straightener.Lift_Entry.Rest := (#Ctrl.EndOfCoil.StraightRollEntry_Open OR #Req OR #TON_Emptying.Q OR #COut.Gen.EmptyingConfirmed) AND NOT #CIn.Straigtener.Lift_Entry.Rest;
   #COut.Straightener.Lift_Entry.Control_ON := NOT (NOT #Sts.Semiautomatic AND NOT #AreaInterface.Cycle AND NOT #TON_Emptying.Q);
END_REGION

REGION Network 98: Coordination Out - Straightener EXIT ROLL
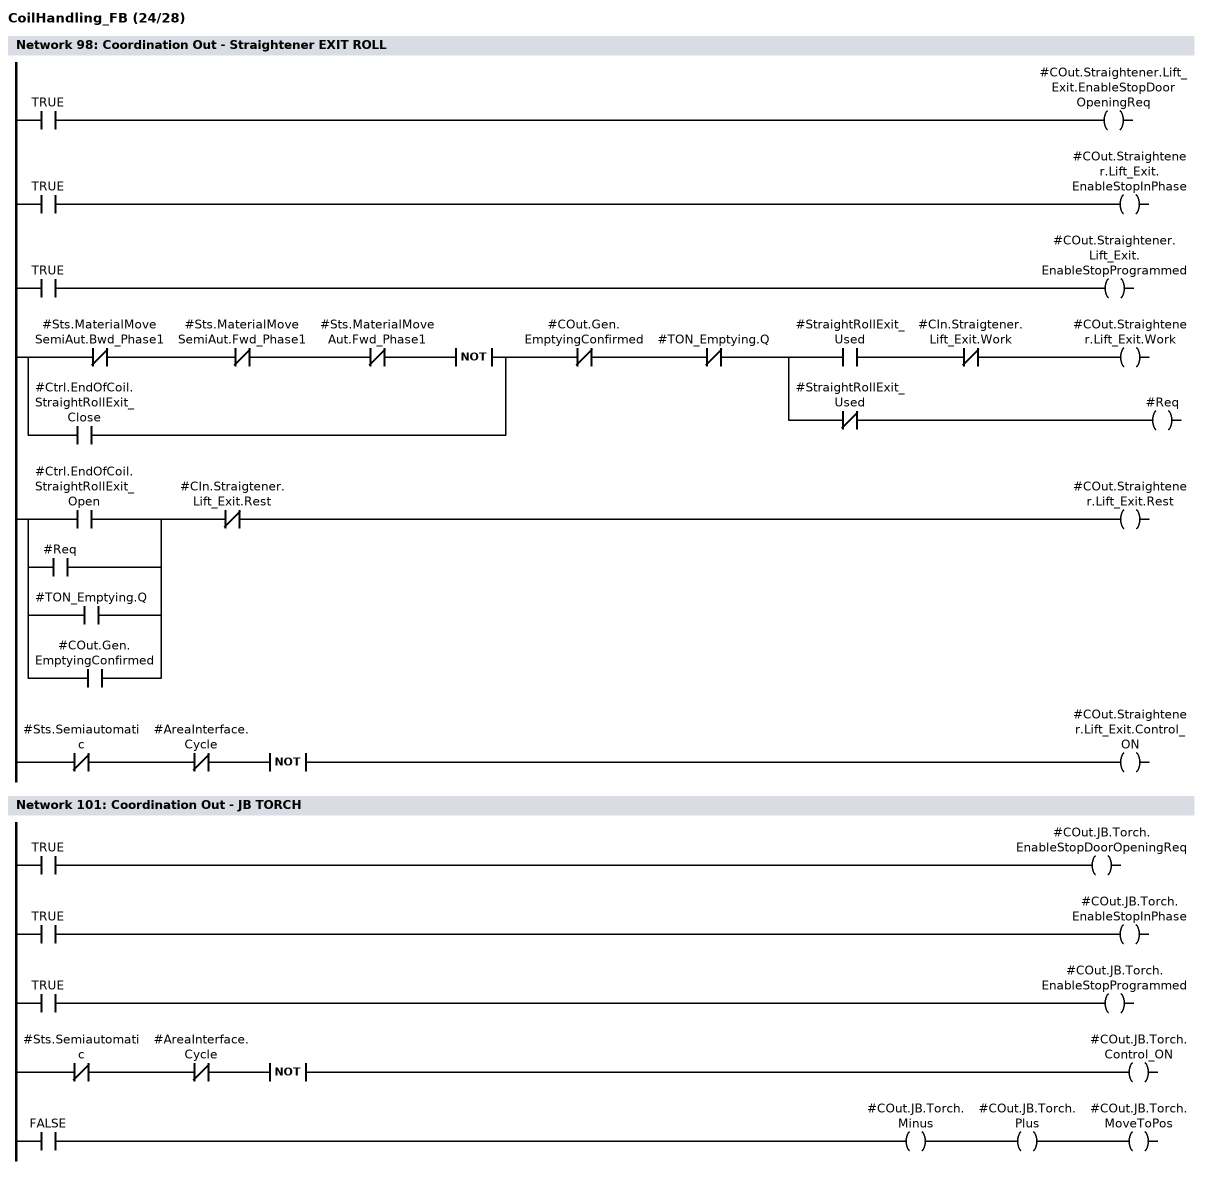
   RUNG wire#powerrail
      Contact( TRUE )
      Coil( #COut.Straightener.Lift_Exit.EnableStopDoorOpeningReq )
   END_RUNG
   RUNG wire#powerrail
      Contact( TRUE )
      Coil( #COut.Straightener.Lift_Exit.EnableStopInPhase )
   END_RUNG
   RUNG wire#powerrail
      Contact( TRUE )
      Coil( #COut.Straightener.Lift_Exit.EnableStopProgrammed )
   END_RUNG
   RUNG wire#powerrail
      I_Contact( #Sts.MaterialMoveSemiAut.Bwd_Phase1 )
      I_Contact( #Sts.MaterialMoveSemiAut.Fwd_Phase1 )
      I_Contact( #Sts.MaterialMoveAut.Fwd_Phase1 )
      Not()
      wire#w1
      I_Contact( #COut.Gen.EmptyingConfirmed )
      I_Contact( #TON_Emptying.Q )
      wire#w2
      Contact( #StraightRollExit_Used )
      I_Contact( #CIn.Straigtener.Lift_Exit.Work )
      Coil( #COut.Straightener.Lift_Exit.Work )
   END_RUNG
   RUNG wire#powerrail
      Contact( #Ctrl.EndOfCoil.StraightRollExit_Close )
   END_RUNG wire#w1
   RUNG wire#w2
      I_Contact( #StraightRollExit_Used )
      Coil( #Req )
   END_RUNG
   RUNG wire#powerrail
      Contact( #Ctrl.EndOfCoil.StraightRollExit_Open )
      wire#w3
      I_Contact( #CIn.Straigtener.Lift_Exit.Rest )
      Coil( #COut.Straightener.Lift_Exit.Rest )
   END_RUNG
   RUNG wire#powerrail
      Contact( #Req )
   END_RUNG wire#w3
   RUNG wire#powerrail
      Contact( #TON_Emptying.Q )
   END_RUNG wire#w3
   RUNG wire#powerrail
      Contact( #COut.Gen.EmptyingConfirmed )
   END_RUNG wire#w3
   RUNG wire#powerrail
      I_Contact( #Sts.Semiautomatic )
      I_Contact( #AreaInterface.Cycle )
      Not()
      Coil( #COut.Straightener.Lift_Exit.Control_ON )
   END_RUNG
   // the same network as SCL:
   #COut.Straightener.Lift_Exit.EnableStopDoorOpeningReq := TRUE;
   #COut.Straightener.Lift_Exit.EnableStopInPhase := TRUE;
   #COut.Straightener.Lift_Exit.EnableStopProgrammed := TRUE;
   #_w1 := (NOT (NOT #Sts.MaterialMoveSemiAut.Bwd_Phase1 AND NOT #Sts.MaterialMoveSemiAut.Fwd_Phase1 AND NOT #Sts.MaterialMoveAut.Fwd_Phase1) OR #Ctrl.EndOfCoil.StraightRollExit_Close) AND NOT #COut.Gen.EmptyingConfirmed AND NOT #TON_Emptying.Q;
   #COut.Straightener.Lift_Exit.Work := #_w1 AND #StraightRollExit_Used AND NOT #CIn.Straigtener.Lift_Exit.Work;
   #Req := #_w1 AND NOT #StraightRollExit_Used;
   #COut.Straightener.Lift_Exit.Rest := (#Ctrl.EndOfCoil.StraightRollExit_Open OR #Req OR #TON_Emptying.Q OR #COut.Gen.EmptyingConfirmed) AND NOT #CIn.Straigtener.Lift_Exit.Rest;
   #COut.Straightener.Lift_Exit.Control_ON := NOT (NOT #Sts.Semiautomatic AND NOT #AreaInterface.Cycle);
END_REGION

REGION Network 99: <+>
END_REGION

REGION Network 100 (SCL): Coordination Out - JB WELDING SET-UP
   #COut.JB.WeldingSetUp.MaterialWidth := "PPrf_MAIN".ON_WORK.GeneralData.Material_Width;
   #COut.JB.WeldingSetUp.MeasureSheetEdgeReference := "PPrf_MAIN".ON_WORK.A01_CoilHandling.WeldingCycle.MeasureSheetEdgeReference;
   #COut.JB.WeldingSetUp.WeldingDirection := TRUE;
   #COut.JB.WeldingSetUp.CorrStartWelding := "PPrf_MAIN".ON_WORK.A01_CoilHandling.WeldingCycle.CorrStartWelding;
   #COut.JB.WeldingSetUp.CorrStopWelding := "PPrf_MAIN".ON_WORK.A01_CoilHandling.WeldingCycle.CorrStopWelding;
END_REGION

REGION Network 101: Coordination Out - JB TORCH
   RUNG wire#powerrail
      Contact( TRUE )
      Coil( #COut.JB.Torch.EnableStopDoorOpeningReq )
   END_RUNG
   RUNG wire#powerrail
      Contact( TRUE )
      Coil( #COut.JB.Torch.EnableStopInPhase )
   END_RUNG
   RUNG wire#powerrail
      Contact( TRUE )
      Coil( #COut.JB.Torch.EnableStopProgrammed )
   END_RUNG
   RUNG wire#powerrail
      I_Contact( #Sts.Semiautomatic )
      I_Contact( #AreaInterface.Cycle )
      Not()
      Coil( #COut.JB.Torch.Control_ON )
   END_RUNG
   RUNG wire#powerrail
      Contact( FALSE )
      Coil( #COut.JB.Torch.Minus )
      Coil( #COut.JB.Torch.Plus )
      Coil( #COut.JB.Torch.MoveToPos )
   END_RUNG
   // the same network as SCL:
   #COut.JB.Torch.EnableStopDoorOpeningReq := TRUE;
   #COut.JB.Torch.EnableStopInPhase := TRUE;
   #COut.JB.Torch.EnableStopProgrammed := TRUE;
   #COut.JB.Torch.Control_ON := NOT (NOT #Sts.Semiautomatic AND NOT #AreaInterface.Cycle);
   #COut.JB.Torch.Minus := FALSE;
   #COut.JB.Torch.Plus := FALSE;
   #COut.JB.Torch.MoveToPos := FALSE;
END_REGION

REGION Network 102: Coordination Out - JB CLAMPS
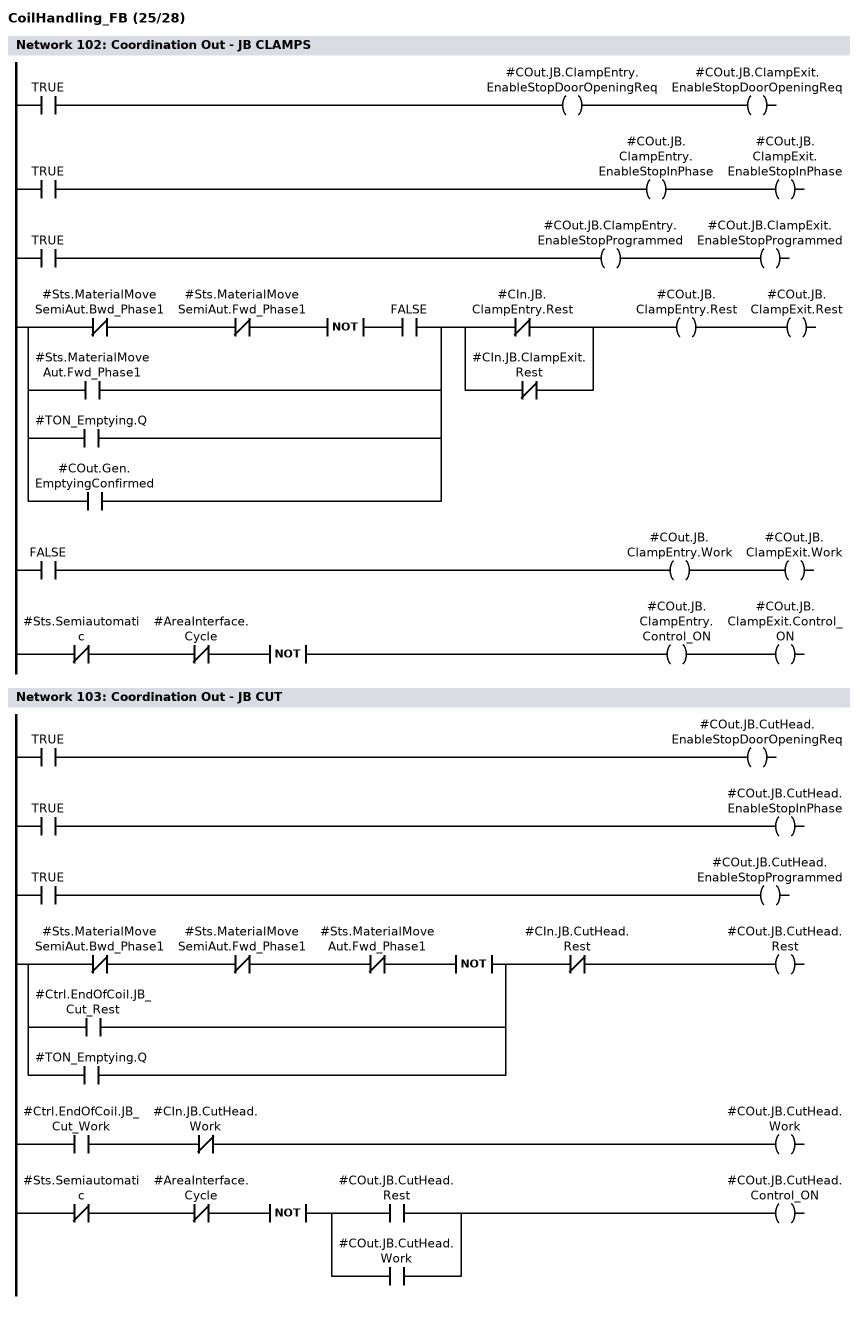
   RUNG wire#powerrail
      Contact( TRUE )
      Coil( #COut.JB.ClampEntry.EnableStopDoorOpeningReq )
      Coil( #COut.JB.ClampExit.EnableStopDoorOpeningReq )
   END_RUNG
   RUNG wire#powerrail
      Contact( TRUE )
      Coil( #COut.JB.ClampEntry.EnableStopInPhase )
      Coil( #COut.JB.ClampExit.EnableStopInPhase )
   END_RUNG
   RUNG wire#powerrail
      Contact( TRUE )
      Coil( #COut.JB.ClampEntry.EnableStopProgrammed )
      Coil( #COut.JB.ClampExit.EnableStopProgrammed )
   END_RUNG
   RUNG wire#powerrail
      I_Contact( #Sts.MaterialMoveSemiAut.Bwd_Phase1 )
      I_Contact( #Sts.MaterialMoveSemiAut.Fwd_Phase1 )
      Not()
      Contact( FALSE )
      wire#w1
      I_Contact( #CIn.JB.ClampEntry.Rest )
      wire#w2
      Coil( #COut.JB.ClampEntry.Rest )
      Coil( #COut.JB.ClampExit.Rest )
   END_RUNG
   RUNG wire#powerrail
      Contact( #Sts.MaterialMoveAut.Fwd_Phase1 )
   END_RUNG wire#w1
   RUNG wire#powerrail
      Contact( #TON_Emptying.Q )
   END_RUNG wire#w1
   RUNG wire#powerrail
      Contact( #COut.Gen.EmptyingConfirmed )
   END_RUNG wire#w1
   RUNG wire#w1
      I_Contact( #CIn.JB.ClampExit.Rest )
   END_RUNG wire#w2
   RUNG wire#powerrail
      Contact( FALSE )
      Coil( #COut.JB.ClampEntry.Work )
      Coil( #COut.JB.ClampExit.Work )
   END_RUNG
   RUNG wire#powerrail
      I_Contact( #Sts.Semiautomatic )
      I_Contact( #AreaInterface.Cycle )
      Not()
      Coil( #COut.JB.ClampEntry.Control_ON )
      Coil( #COut.JB.ClampExit.Control_ON )
   END_RUNG
   // the same network as SCL:
   #COut.JB.ClampEntry.EnableStopDoorOpeningReq := TRUE;
   #COut.JB.ClampExit.EnableStopDoorOpeningReq := TRUE;
   #COut.JB.ClampEntry.EnableStopInPhase := TRUE;
   #COut.JB.ClampExit.EnableStopInPhase := TRUE;
   #COut.JB.ClampEntry.EnableStopProgrammed := TRUE;
   #COut.JB.ClampExit.EnableStopProgrammed := TRUE;
   #COut.JB.ClampEntry.Rest := ((NOT (NOT #Sts.MaterialMoveSemiAut.Bwd_Phase1 AND NOT #Sts.MaterialMoveSemiAut.Fwd_Phase1) AND FALSE) OR #Sts.MaterialMoveAut.Fwd_Phase1 OR #TON_Emptying.Q OR #COut.Gen.EmptyingConfirmed) AND (NOT #CIn.JB.ClampEntry.Rest OR NOT #CIn.JB.ClampExit.Rest);
   #COut.JB.ClampExit.Rest := #COut.JB.ClampEntry.Rest;
   #COut.JB.ClampEntry.Work := FALSE;
   #COut.JB.ClampExit.Work := FALSE;
   #COut.JB.ClampEntry.Control_ON := NOT (NOT #Sts.Semiautomatic AND NOT #AreaInterface.Cycle);
   #COut.JB.ClampExit.Control_ON := #COut.JB.ClampEntry.Control_ON;
END_REGION

REGION Network 103: Coordination Out - JB CUT
   RUNG wire#powerrail
      Contact( TRUE )
      Coil( #COut.JB.CutHead.EnableStopDoorOpeningReq )
   END_RUNG
   RUNG wire#powerrail
      Contact( TRUE )
      Coil( #COut.JB.CutHead.EnableStopInPhase )
   END_RUNG
   RUNG wire#powerrail
      Contact( TRUE )
      Coil( #COut.JB.CutHead.EnableStopProgrammed )
   END_RUNG
   RUNG wire#powerrail
      I_Contact( #Sts.MaterialMoveSemiAut.Bwd_Phase1 )
      I_Contact( #Sts.MaterialMoveSemiAut.Fwd_Phase1 )
      I_Contact( #Sts.MaterialMoveAut.Fwd_Phase1 )
      Not()
      wire#w1
      I_Contact( #CIn.JB.CutHead.Rest )
      Coil( #COut.JB.CutHead.Rest )
   END_RUNG
   RUNG wire#powerrail
      Contact( #Ctrl.EndOfCoil.JB_Cut_Rest )
   END_RUNG wire#w1
   RUNG wire#powerrail
      Contact( #TON_Emptying.Q )
   END_RUNG wire#w1
   RUNG wire#powerrail
      Contact( #Ctrl.EndOfCoil.JB_Cut_Work )
      I_Contact( #CIn.JB.CutHead.Work )
      Coil( #COut.JB.CutHead.Work )
   END_RUNG
   RUNG wire#powerrail
      I_Contact( #Sts.Semiautomatic )
      I_Contact( #AreaInterface.Cycle )
      Not()
      wire#w2
      Contact( #COut.JB.CutHead.Rest )
      wire#w3
      Coil( #COut.JB.CutHead.Control_ON )
   END_RUNG
   RUNG wire#w2
      Contact( #COut.JB.CutHead.Work )
   END_RUNG wire#w3
   // the same network as SCL:
   #COut.JB.CutHead.EnableStopDoorOpeningReq := TRUE;
   #COut.JB.CutHead.EnableStopInPhase := TRUE;
   #COut.JB.CutHead.EnableStopProgrammed := TRUE;
   #COut.JB.CutHead.Rest := (NOT (NOT #Sts.MaterialMoveSemiAut.Bwd_Phase1 AND NOT #Sts.MaterialMoveSemiAut.Fwd_Phase1 AND NOT #Sts.MaterialMoveAut.Fwd_Phase1) OR #Ctrl.EndOfCoil.JB_Cut_Rest OR #TON_Emptying.Q) AND NOT #CIn.JB.CutHead.Rest;
   #COut.JB.CutHead.Work := #Ctrl.EndOfCoil.JB_Cut_Work AND NOT #CIn.JB.CutHead.Work;
   #COut.JB.CutHead.Control_ON := NOT (NOT #Sts.Semiautomatic AND NOT #AreaInterface.Cycle) AND (#COut.JB.CutHead.Rest OR #COut.JB.CutHead.Work);
END_REGION

REGION Network 104: Coordination Out - JB Pinch roll FEED
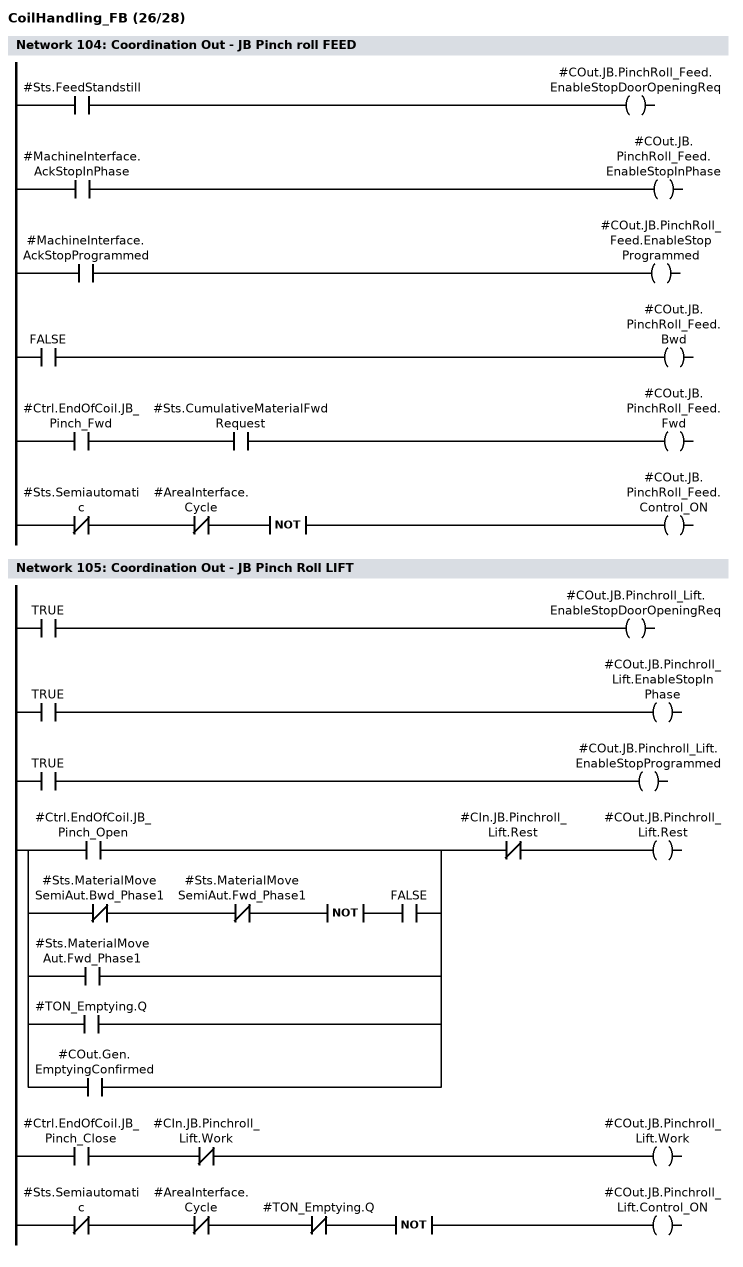
   RUNG wire#powerrail
      Contact( #Sts.FeedStandstill )
      Coil( #COut.JB.PinchRoll_Feed.EnableStopDoorOpeningReq )
   END_RUNG
   RUNG wire#powerrail
      Contact( #MachineInterface.AckStopInPhase )
      Coil( #COut.JB.PinchRoll_Feed.EnableStopInPhase )
   END_RUNG
   RUNG wire#powerrail
      Contact( #MachineInterface.AckStopProgrammed )
      Coil( #COut.JB.PinchRoll_Feed.EnableStopProgrammed )
   END_RUNG
   RUNG wire#powerrail
      Contact( FALSE )
      Coil( #COut.JB.PinchRoll_Feed.Bwd )
   END_RUNG
   RUNG wire#powerrail
      Contact( #Ctrl.EndOfCoil.JB_Pinch_Fwd )
      Contact( #Sts.CumulativeMaterialFwdRequest )
      Coil( #COut.JB.PinchRoll_Feed.Fwd )
   END_RUNG
   RUNG wire#powerrail
      I_Contact( #Sts.Semiautomatic )
      I_Contact( #AreaInterface.Cycle )
      Not()
      Coil( #COut.JB.PinchRoll_Feed.Control_ON )
   END_RUNG
   // the same network as SCL:
   #COut.JB.PinchRoll_Feed.EnableStopDoorOpeningReq := #Sts.FeedStandstill;
   #COut.JB.PinchRoll_Feed.EnableStopInPhase := #MachineInterface.AckStopInPhase;
   #COut.JB.PinchRoll_Feed.EnableStopProgrammed := #MachineInterface.AckStopProgrammed;
   #COut.JB.PinchRoll_Feed.Bwd := FALSE;
   #COut.JB.PinchRoll_Feed.Fwd := #Ctrl.EndOfCoil.JB_Pinch_Fwd AND #Sts.CumulativeMaterialFwdRequest;
   #COut.JB.PinchRoll_Feed.Control_ON := NOT (NOT #Sts.Semiautomatic AND NOT #AreaInterface.Cycle);
END_REGION

REGION Network 105: Coordination Out - JB Pinch Roll LIFT
   RUNG wire#powerrail
      Contact( TRUE )
      Coil( #COut.JB.Pinchroll_Lift.EnableStopDoorOpeningReq )
   END_RUNG
   RUNG wire#powerrail
      Contact( TRUE )
      Coil( #COut.JB.Pinchroll_Lift.EnableStopInPhase )
   END_RUNG
   RUNG wire#powerrail
      Contact( TRUE )
      Coil( #COut.JB.Pinchroll_Lift.EnableStopProgrammed )
   END_RUNG
   RUNG wire#powerrail
      Contact( #Ctrl.EndOfCoil.JB_Pinch_Open )
      wire#w1
      I_Contact( #CIn.JB.Pinchroll_Lift.Rest )
      Coil( #COut.JB.Pinchroll_Lift.Rest )
   END_RUNG
   RUNG wire#powerrail
      I_Contact( #Sts.MaterialMoveSemiAut.Bwd_Phase1 )
      I_Contact( #Sts.MaterialMoveSemiAut.Fwd_Phase1 )
      Not()
      Contact( FALSE )
   END_RUNG wire#w1
   RUNG wire#powerrail
      Contact( #Sts.MaterialMoveAut.Fwd_Phase1 )
   END_RUNG wire#w1
   RUNG wire#powerrail
      Contact( #TON_Emptying.Q )
   END_RUNG wire#w1
   RUNG wire#powerrail
      Contact( #COut.Gen.EmptyingConfirmed )
   END_RUNG wire#w1
   RUNG wire#powerrail
      Contact( #Ctrl.EndOfCoil.JB_Pinch_Close )
      I_Contact( #CIn.JB.Pinchroll_Lift.Work )
      Coil( #COut.JB.Pinchroll_Lift.Work )
   END_RUNG
   RUNG wire#powerrail
      I_Contact( #Sts.Semiautomatic )
      I_Contact( #AreaInterface.Cycle )
      I_Contact( #TON_Emptying.Q )
      Not()
      Coil( #COut.JB.Pinchroll_Lift.Control_ON )
   END_RUNG
   // the same network as SCL:
   #COut.JB.Pinchroll_Lift.EnableStopDoorOpeningReq := TRUE;
   #COut.JB.Pinchroll_Lift.EnableStopInPhase := TRUE;
   #COut.JB.Pinchroll_Lift.EnableStopProgrammed := TRUE;
   #COut.JB.Pinchroll_Lift.Rest := (#Ctrl.EndOfCoil.JB_Pinch_Open OR (NOT (NOT #Sts.MaterialMoveSemiAut.Bwd_Phase1 AND NOT #Sts.MaterialMoveSemiAut.Fwd_Phase1) AND FALSE) OR #Sts.MaterialMoveAut.Fwd_Phase1 OR #TON_Emptying.Q OR #COut.Gen.EmptyingConfirmed) AND NOT #CIn.JB.Pinchroll_Lift.Rest;
   #COut.JB.Pinchroll_Lift.Work := #Ctrl.EndOfCoil.JB_Pinch_Close AND NOT #CIn.JB.Pinchroll_Lift.Work;
   #COut.JB.Pinchroll_Lift.Control_ON := NOT (NOT #Sts.Semiautomatic AND NOT #AreaInterface.Cycle AND NOT #TON_Emptying.Q);
END_REGION

REGION Network 106: <+>
END_REGION

REGION Network 107: <+>
END_REGION

REGION Network 108: Coordination Out - Loop 1
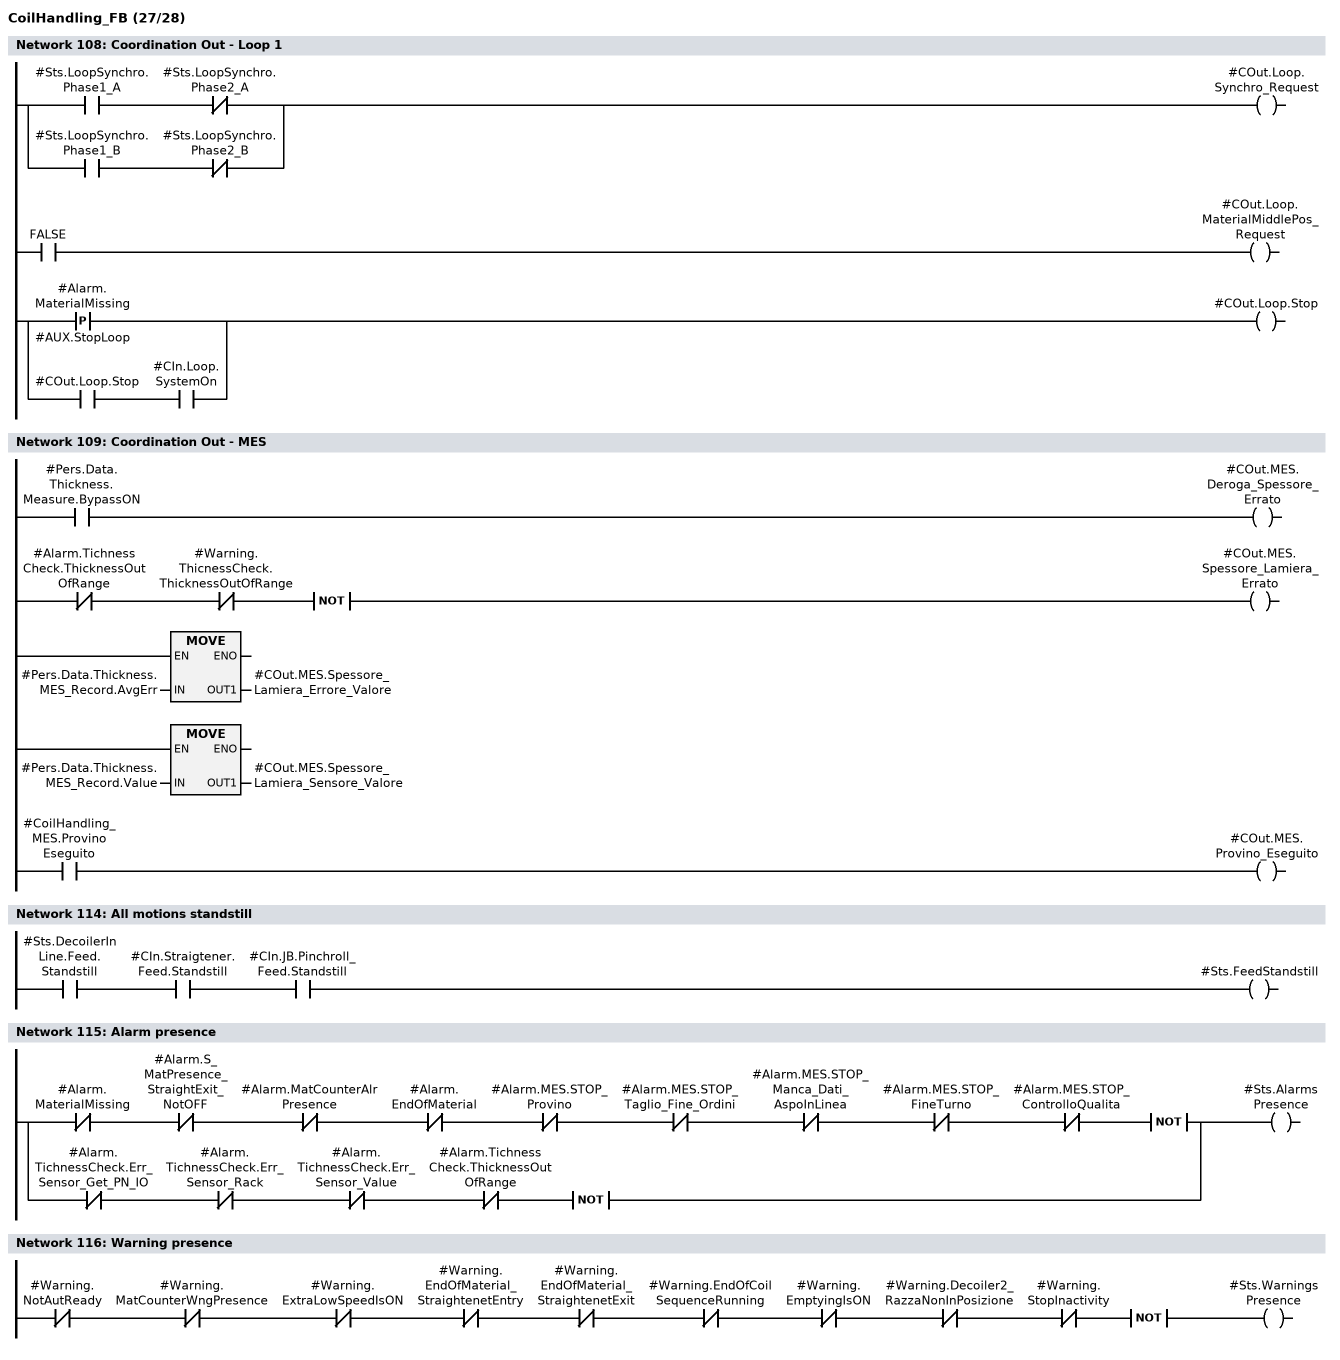
   RUNG wire#powerrail
      Contact( #Sts.LoopSynchro.Phase1_A )
      I_Contact( #Sts.LoopSynchro.Phase2_A )
      wire#w1
      Coil( #COut.Loop.Synchro_Request )
   END_RUNG
   RUNG wire#powerrail
      Contact( #Sts.LoopSynchro.Phase1_B )
      I_Contact( #Sts.LoopSynchro.Phase2_B )
   END_RUNG wire#w1
   RUNG wire#powerrail
      Contact( FALSE )
      Coil( #COut.Loop.MaterialMiddlePos_Request )
   END_RUNG
   RUNG wire#powerrail
      P_Contact(operand := #Alarm.MaterialMissing, bit := #AUX.StopLoop)
      wire#w2
      Coil( #COut.Loop.Stop )
   END_RUNG
   RUNG wire#powerrail
      Contact( #COut.Loop.Stop )
      Contact( #CIn.Loop.SystemOn )
   END_RUNG wire#w2
   // the same network as SCL:
   #COut.Loop.Synchro_Request := (#Sts.LoopSynchro.Phase1_A AND NOT #Sts.LoopSynchro.Phase2_A) OR (#Sts.LoopSynchro.Phase1_B AND NOT #Sts.LoopSynchro.Phase2_B);
   #COut.Loop.MaterialMiddlePos_Request := FALSE;
   #_w1 := #Alarm.MaterialMissing AND NOT #AUX.StopLoop;   // rising edge of #Alarm.MaterialMissing
   #AUX.StopLoop := #Alarm.MaterialMissing;
   #COut.Loop.Stop := #_w1 OR (#COut.Loop.Stop AND #CIn.Loop.SystemOn);
END_REGION

REGION Network 109: Coordination Out - MES
   RUNG wire#powerrail
      Contact( #Pers.Data.Thickness.Measure.BypassON )
      Coil( #COut.MES.Deroga_Spessore_Errato )
   END_RUNG
   RUNG wire#powerrail
      I_Contact( #Alarm.TichnessCheck.ThicknessOutOfRange )
      I_Contact( #Warning.ThicnessCheck.ThicknessOutOfRange )
      Not()
      Coil( #COut.MES.Spessore_Lamiera_Errato )
   END_RUNG
   RUNG wire#powerrail
      Move(in := #Pers.Data.Thickness.MES_Record.AvgErr, out1 => #COut.MES.Spessore_Lamiera_Errore_Valore)
   END_RUNG
   RUNG wire#powerrail
      Move(in := #Pers.Data.Thickness.MES_Record.Value, out1 => #COut.MES.Spessore_Lamiera_Sensore_Valore)
   END_RUNG
   RUNG wire#powerrail
      Contact( #CoilHandling_MES.ProvinoEseguito )
      Coil( #COut.MES.Provino_Eseguito )
   END_RUNG
   // the same network as SCL:
   #COut.MES.Deroga_Spessore_Errato := #Pers.Data.Thickness.Measure.BypassON;
   #COut.MES.Spessore_Lamiera_Errato := NOT (NOT #Alarm.TichnessCheck.ThicknessOutOfRange AND NOT #Warning.ThicnessCheck.ThicknessOutOfRange);
   #COut.MES.Spessore_Lamiera_Errore_Valore := #Pers.Data.Thickness.MES_Record.AvgErr;
   #COut.MES.Spessore_Lamiera_Sensore_Valore := #Pers.Data.Thickness.MES_Record.Value;
   #COut.MES.Provino_Eseguito := #CoilHandling_MES.ProvinoEseguito;
END_REGION

REGION Network 110: >
END_REGION

REGION Network 111: >
END_REGION

REGION Network 112: >
END_REGION

REGION Network 113: << FINAL OPERATIONS >>
   // +
   // +
   // +
   // +
   // +
   // +
   // +
   // +
   // +
   // +
   // +
   // +
   // +
END_REGION

REGION Network 114: All motions standstill
   RUNG wire#powerrail
      Contact( #Sts.DecoilerInLine.Feed.Standstill )
      Contact( #CIn.Straigtener.Feed.Standstill )
      Contact( #CIn.JB.Pinchroll_Feed.Standstill )
      Coil( #Sts.FeedStandstill )
   END_RUNG
   // the same network as SCL:
   #Sts.FeedStandstill := #Sts.DecoilerInLine.Feed.Standstill AND #CIn.Straigtener.Feed.Standstill AND #CIn.JB.Pinchroll_Feed.Standstill;
END_REGION

REGION Network 115: Alarm presence
   RUNG wire#powerrail
      I_Contact( #Alarm.MaterialMissing )
      I_Contact( #Alarm.S_MatPresence_StraightExit_NotOFF )
      I_Contact( #Alarm.MatCounterAlrPresence )
      I_Contact( #Alarm.EndOfMaterial )
      I_Contact( #Alarm.MES.STOP_Provino )
      I_Contact( #Alarm.MES.STOP_Taglio_Fine_Ordini )
      I_Contact( #Alarm.MES.STOP_Manca_Dati_AspoInLinea )
      I_Contact( #Alarm.MES.STOP_FineTurno )
      I_Contact( #Alarm.MES.STOP_ControlloQualita )
      Not()
      wire#w1
      Coil( #Sts.AlarmsPresence )
   END_RUNG
   RUNG wire#powerrail
      I_Contact( #Alarm.TichnessCheck.Err_Sensor_Get_PN_IO )
      I_Contact( #Alarm.TichnessCheck.Err_Sensor_Rack )
      I_Contact( #Alarm.TichnessCheck.Err_Sensor_Value )
      I_Contact( #Alarm.TichnessCheck.ThicknessOutOfRange )
      Not()
   END_RUNG wire#w1
   // the same network as SCL:
   #Sts.AlarmsPresence := NOT (NOT #Alarm.MaterialMissing AND NOT #Alarm.S_MatPresence_StraightExit_NotOFF AND NOT #Alarm.MatCounterAlrPresence AND NOT #Alarm.EndOfMaterial AND NOT #Alarm.MES.STOP_Provino AND NOT #Alarm.MES.STOP_Taglio_Fine_Ordini AND NOT #Alarm.MES.STOP_Manca_Dati_AspoInLinea AND NOT #Alarm.MES.STOP_FineTurno AND NOT #Alarm.MES.STOP_ControlloQualita) OR NOT (NOT #Alarm.TichnessCheck.Err_Sensor_Get_PN_IO AND NOT #Alarm.TichnessCheck.Err_Sensor_Rack AND NOT #Alarm.TichnessCheck.Err_Sensor_Value AND NOT #Alarm.TichnessCheck.ThicknessOutOfRange);
END_REGION

REGION Network 116: Warning presence
   RUNG wire#powerrail
      I_Contact( #Warning.NotAutReady )
      I_Contact( #Warning.MatCounterWngPresence )
      I_Contact( #Warning.ExtraLowSpeedIsON )
      I_Contact( #Warning.EndOfMaterial_StraightenetEntry )
      I_Contact( #Warning.EndOfMaterial_StraightenetExit )
      I_Contact( #Warning.EndOfCoilSequenceRunning )
      I_Contact( #Warning.EmptyingIsON )
      I_Contact( #Warning.Decoiler2_RazzaNonInPosizione )
      I_Contact( #Warning.StopInactivity )
      Not()
      Coil( #Sts.WarningsPresence )
   END_RUNG
   // the same network as SCL:
   #Sts.WarningsPresence := NOT (NOT #Warning.NotAutReady AND NOT #Warning.MatCounterWngPresence AND NOT #Warning.ExtraLowSpeedIsON AND NOT #Warning.EndOfMaterial_StraightenetEntry AND NOT #Warning.EndOfMaterial_StraightenetExit AND NOT #Warning.EndOfCoilSequenceRunning AND NOT #Warning.EmptyingIsON AND NOT #Warning.Decoiler2_RazzaNonInPosizione AND NOT #Warning.StopInactivity);
END_REGION

REGION Network 117 (SCL): Collect machine to area interface
   #MachineInterface.AutReady := #AreaInterface.Aut AND NOT #Sts.AlarmsPresence;

   #MachineInterface.MotionsStandStill := #Sts.FeedStandstill ;

   // Status machine aborting
   #MachineInterface.Aborting := #Ctrl.Stop AND #MachineInterface.MotionsStandStill;

   // Status Ack Stop in phase
   #MachineInterface.AckStopInPhase := #AreaInterface.StopInPhase AND #MachineInterface.MotionsStandStill;
   // Status Ack Stop programmed
   #MachineInterface.AckStopProgrammed := #AreaInterface.StopProgrammed AND #MachineInterface.MotionsStandStill;

   // Status Alarm presence
   #MachineInterface.AlarmsPresence := #Sts.AlarmsPresence;
   // Status Warning presence
   #MachineInterface.WarningPresence := #Sts.WarningsPresence;
END_REGION

REGION Network 118: Warning Machine not ready for automatic
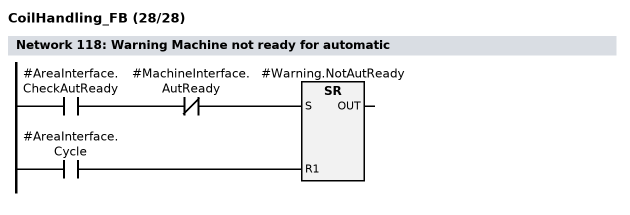
   RUNG wire#powerrail
      Contact( #AreaInterface.CheckAutReady )
      I_Contact( #MachineInterface.AutReady )
      S_SR(operand := #Warning.NotAutReady, r1 := wire#w1)
   END_RUNG
   RUNG wire#powerrail
      Contact( #AreaInterface.Cycle )
   END_RUNG wire#w1
   // the same network as SCL:
   IF #AreaInterface.CheckAutReady AND NOT #MachineInterface.AutReady THEN
       #Warning.NotAutReady := TRUE;   // SR flip-flop
   END_IF;
   IF #AreaInterface.Cycle THEN #Warning.NotAutReady := FALSE; END_IF;
END_REGION

REGION Network 119 (SCL): ENO
   ENO := NOT #Sts.AlarmsPresence;
END_REGION
END_FUNCTION_BLOCK
